FUNCTION_BLOCK CmdWaterDischargeSLB (* CAT Function Block Type *)
  (* Standard: 61499-2 *)
  (* Version 2.0, 10/1/2026, Claude/Hidryco, Schneider Electric, Rev2 - Cmin (velocidade minima por bomba) do IThis para a logica; Rev1 - Nivel L e pausa (T_Restart/T_FlowLL); Modo sobrenadante (2 servico + 1 reserva); parametros Cmax/C2/C3/T_C2/T_C3; LOAD_PERS_DATA na inicializacao *)
  PACKAGE SE.Nereda;
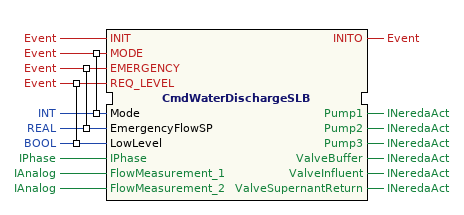
  EVENT_INPUT
    INIT;
    MODE WITH Mode;
    EMERGENCY WITH EmergencyFlowSP;
    REQ_LEVEL WITH LowLevel; (* Nivel L do 49LT0001 *)
  END_EVENT
  EVENT_OUTPUT
    INITO;
  END_EVENT
  VAR_INPUT
    Mode : INT;
    EmergencyFlowSP : REAL;
    LowLevel : BOOL; (* Nivel L do 49LT0001 (pausa a descarga) *)
  END_VAR
  SOCKETS
    IPhase : IPhase;
  END_SOCKETS
  SOCKETS
    FlowMeasurement_1 : IAnalog;
    FlowMeasurement_2 : IAnalog;
  END_SOCKETS
  PLUGS
    Pump1 : INeredaAct;
    Pump2 : INeredaAct;
    Pump3 : INeredaAct;
    ValveBuffer : INeredaAct;
    ValveInfluent : INeredaAct;
    ValveSupernantReturn : INeredaAct;
  END_PLUGS
  (* 01 - FUNCTIONNAL INPUT INTERFACE *)
  (* 00 - INITIALIZATION *)
  (* 05 - LOGIC *)
  (* 06 - HMI INTERFACE *)
  (* 03 - FIELD INTERFACE *)
  (* 02 - FUNCTIONNAL OUTPUT INTERFACE *)
  (* Command Logic *)
  (* Capacity Setpoint *)
  FBS
    IThis : CmdWaterDischargeSLB_HMI(QI := TRUE);
    FeedFlowSpParameterSelector : ParametersSelector;
    CommandLogic : CmdSludgeDischargeSLBLogic(pin_EDA46437701491D7 := TRUE); {SET_ATTRIBUTE(Configuration.Component.HideUnusedPorts, )}
  END_FBS
  EVENT_CONNECTIONS
    MODE TO FeedFlowSpParameterSelector.MODE;
    EMERGENCY TO FeedFlowSpParameterSelector.3B878B7E006C38E4;
    INIT TO IThis.C4758748B8B7D3EA;
    IThis.851B32D559A6AA3F TO FeedFlowSpParameterSelector.REQ_NEREDA_VAL;
    IThis.59FB590F9F8A710E TO FeedFlowSpParameterSelector.REQ_MAN_VAL;
    IPhase.Interlocked_CNF TO CommandLogic.393B564B9DA2DBA7;
    FeedFlowSpParameterSelector.CNF TO CommandLogic.971F31261154ACD5;
    IThis.9FEA1874A72DD629 TO CommandLogic.A14398C211A20C12;
    CommandLogic.75C95E56F6162690 TO INITO;
    CommandLogic.3441D16350C1D291 TO IPhase.REQ_Start_Ready;
    CommandLogic.C8B1A85D0153CD87 TO IPhase.REQ_Stop_Ready;
    CommandLogic.53236A8C814FFA4F TO IPhase.REQ_Abort_Ready;
    IThis.5057011FA5ED4FF7 TO CommandLogic.65CF25B02F3B6C57;
    CommandLogic.75C95E56F6162690 TO IThis.E235583F49B9570B;
    REQ_LEVEL TO CommandLogic.024991AC33B2DF2D;
    IThis.F5A96D7EEB24B101 TO CommandLogic.65CF25B02F3B6C57;
    IThis.5F8E6D9D33956FD6 TO CommandLogic.65CF25B02F3B6C57;
  END_CONNECTIONS
  DATA_CONNECTIONS
    Mode TO FeedFlowSpParameterSelector.Mode;
    EmergencyFlowSP TO FeedFlowSpParameterSelector.4C6C1BFF70182CBB;
    IThis.48FC57B4BA0AB67A TO FeedFlowSpParameterSelector.NeredaValue;
    IThis.C4072BA96C21EBC0 TO FeedFlowSpParameterSelector.ManValue;
    IPhase.Ready TO CommandLogic.C1328A46AF65D0A6;
    IPhase.Starting TO CommandLogic.B6C61BC7391E4616;
    IPhase.Run TO CommandLogic.8259B159B326D7FF;
    IPhase.Stopping TO CommandLogic.B7C1C59879F9DA01;
    IPhase.Aborting TO CommandLogic.308AFE103F900E24;
    FeedFlowSpParameterSelector.ValOut TO CommandLogic.D65A4A7591488987;
    CommandLogic.A0873A10F64BE3F2 TO IPhase.Start_Ready;
    CommandLogic.3E5CE56C6D257D11 TO IPhase.Stop_Ready;
    CommandLogic.3EC99F3974DE065F TO IPhase.Abort_Ready;
    IThis.9EE8317B8E069AB0 TO CommandLogic.9743FA817FB33581;
    IThis.9780816DAABEA3AC TO CommandLogic.9E4EFA5F05462127;
    IThis.186FFB4FD796086C TO CommandLogic.80864F97B82059EB;
    IThis.7C24DA33FAF6C65C TO CommandLogic.59DAA3F863258147;
    IThis.932C418507DF85D3 TO CommandLogic.443B51A39FD2F517;
    LowLevel TO CommandLogic.0F129CC61BF3460D;
    IThis.409925CDAB4F13AD TO CommandLogic.26D3C3E31EC21607;
    IThis.D39553B54E329FDF TO CommandLogic.22E149C0CC432615;
    IThis.A932B147BEA14658 TO CommandLogic.A13D37C90CBA8B2D;
  END_CONNECTIONS
  ADAPTER_CONNECTIONS
    FlowMeasurement_1 TO CommandLogic.F89AF997F6D64559;
    FlowMeasurement_2 TO CommandLogic.4CB774539D1540E0;
    CommandLogic.4472550908FB2BBA TO Pump1;
    CommandLogic.E69CD644C3AB364B TO Pump2;
    CommandLogic.80FEDED2D558DFFC TO Pump3;
    CommandLogic.1FE182D7291AACCE TO ValveBuffer;
    CommandLogic.6243C1FB70DE9E92 TO ValveInfluent;
    CommandLogic.56E89BA7A8737F32 TO ValveSupernantReturn;
  END_CONNECTIONS
END_FUNCTION_BLOCK
